TYPE "MEStoPLC_RecipeData_OP220"
VERSION : 0.1
   STRUCT
      "M-PartType" : String[28];
      "M-PartTypeRecordNr" : Int;
      "M-RecipeVer" : String[18];
      "M-RecipeParameter" { S7_SetPoint := 'False'} : "MEStoPLC_RecipeParameter_OP220";
      Reserve : Array[1..1436] of Byte;
   END_STRUCT;

END_TYPE

